ABB RobotStudio station: P2_Nueva_Ejercicio2_1.rsstnx

Station P2_Nueva_Ejercicio1 (saved by RobotStudio 24.4.11080.0)
Controller Controlador1
  mechanical unit ROB_1: IRB1200_5_90_STD_03, 6 joints, base frame (0, 0, 0) mm
Layout (positions relative to the parent item):
  - IRB1200_5_90_STD_03 [mechanism, from %ABB.RobotStudio.Models.IRB1200%\IRB1200_5_90_STD_03.rslib] at (0, 0, 0) mm; joint values [0, 0, 0, 0, 0.5236, 0] (rad or m)
  - MyTool [mechanism, from Training Objects\myTool.rslib] at (522.01, 0, 848.1) mm, rotated rx 180 ry 60 rz 180 deg
  - Pieza_1 [part] at (-108.51, -174.2, 0) mm, size 669.6 x 559.8 x 200 mm
Attachment: MyTool is attached to IRB1200_5_90_STD_03 / Link6
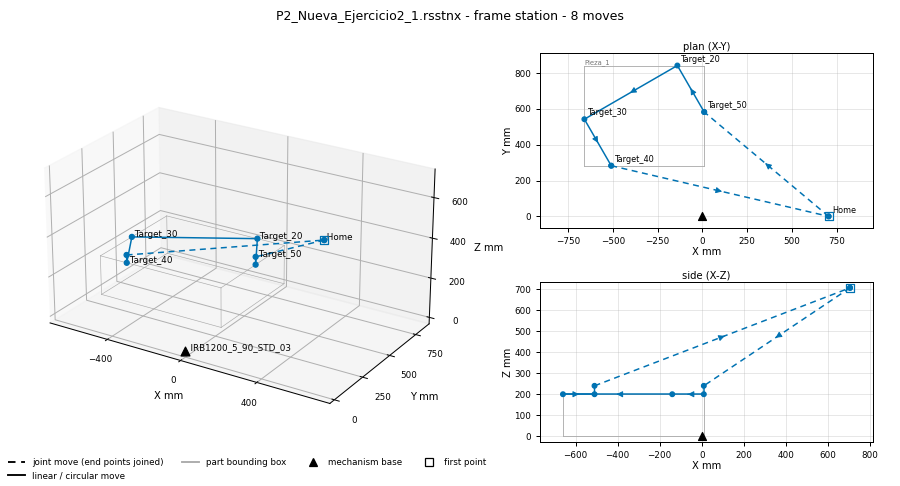
[picture p0: tool path of P2_Nueva_Ejercicio2_1.rsstnx in frame station, 8 of 8 moves have a stored position in this frame; points joined in program order, loops and branches not executed]
Targets, tools, work objects and paths stored in the station, written as RAPID:
! task T_ROB1
MODULE CalibData
  PERS tooldata MyTool:=[TRUE,[[31.792631019,0,229.638935148],[0.945518576,0,0.325568154,0]],[1,[0,0,1],[1,0,0,0],0,0,0]];
  TASK PERS wobjdata WO_Caja:=[FALSE,TRUE,"",[[-140.192,842.82,0],[0.5,0,0,0.866025404]],[[0,0,0],[1,0,0,0]]];
ENDMODULE

! task T_ROB1
MODULE Module1
  CONST robtarget Home:=[[704.990919137,0,705.74730631],[0.190808996,0,0.981627183,0],[0,0,0,0],[9E+09,9E+09,9E+09,9E+09,9E+09,9E+09]];
  CONST robtarget Target_10:=[[-300,0,200],[0,0,1,0],[-1,0,-2,0],[9E+09,9E+09,9E+09,9E+09,9E+09,9E+09]];
  CONST robtarget Target_20:=[[0,0,200],[0,0,1,0],[1,0,-1,0],[9E+09,9E+09,9E+09,9E+09,9E+09,9E+09]];
  CONST robtarget Target_30:=[[0,600,200],[0,0,1,0],[1,-1,0,0],[9E+09,9E+09,9E+09,9E+09,9E+09,9E+09]];
  CONST robtarget Target_40:=[[-300,600,200],[0,0,1,0],[0,-1,1,0],[9E+09,9E+09,9E+09,9E+09,9E+09,9E+09]];
  CONST robtarget Target_50:=[[-299.999462081,-0.000310503,240],[0,0,1,0],[0,0,-2,0],[9E+09,9E+09,9E+09,9E+09,9E+09,9E+09]];
  CONST robtarget Target_60:=[[-299.999083087,600.00034571,240],[0,0,1,0],[1,-1,1,0],[9E+09,9E+09,9E+09,9E+09,9E+09,9E+09]];
  PROC Perimetro_caja()
    MoveL Home,v200,fine,MyTool\WObj:=wobj0;
    MoveJ Target_50,v200,fine,MyTool\WObj:=WO_Caja;
    MoveL Target_10,v200,fine,MyTool\WObj:=WO_Caja;
    MoveL Target_20,v200,fine,MyTool\WObj:=WO_Caja;
    MoveL Target_30,v200,fine,MyTool\WObj:=WO_Caja;
    MoveL Target_40,v200,fine,MyTool\WObj:=WO_Caja;
    MoveL Target_60,v200,fine,MyTool\WObj:=WO_Caja;
    MoveJ Home,v200,fine,MyTool\WObj:=wobj0;
  ENDPROC
ENDMODULE

